PROGRAM PRG1_Conveyer_Operation
VAR_INPUT
	
END_VAR
VAR
	weegTijd 			: INT 			:= 0;
	weegEind 			: INT 			:= 50;
	runningTijd  		: INT 			:= 0;
	detectieLaagTijd  	: INT 			:= 40;
	alarmTijd			: INT			:= 0;
	Modus				: STRING(INT#8) := 'OFF';
	voortangDeling		: INT			:= 100;
	checkpunt			: INT 			:= 0;
END_VAR


// Read startknop
IF NOT GVL.KN_001 AND NOT GVL.alarmActief THEN
	GVL.PRG1_Status := 0;
	GVL.transportActief := FALSE;
END_IF

//als alarm dan naar FAULT
IF NOT GVL.KN_001 AND GVL.alarmActief THEN
	GVL.PRG1_Status := 3;
END_IF

//case functie, voor conveyerstatussen
CASE GVL.PRG1_Status OF
	0:	// OFF, wacht op startknop
		Modus := 'OFF';
		
		IF GVL.KN_001 THEN
			GVL.PRG1_Status := 1;
		END_IF
	1: // idle, wacht op object	
		Modus := 'IDLE';
		
		//reset berekening voor volgende weging
		GVL.berekendeSnelheid := 0;
		
		// als no object detected berekent FC1 de maximale tijd tot alarm
		IF GVL.objectDetected = TRUE THEN
			
			weegTijd := weegTijd + 2;
			GVL.ladingGewicht := GVL.weegcelWaarde;								
			GVL.berekendeSnelheid := FC1_Bereken_Snelheid(GVL.ladingGewicht);//GVL.MinGewicht, GVL.MaxGewicht,GVL.MinSpeed,GVL.MaxSpeed
			IF weegTijd >= weegEind THEN
				GVL.PRG1_Status := 2;
				//reset weegtijd
				weegTijd := 0;
			END_IF
			
		END_IF
		
	2: //running
		Modus := 'RUNNING';
		
		GVL.transportActief := TRUE;
		GVL.geschrevenSnelheid := GVL.berekendeSnelheid;
			
		// Runtijd tellen
		runningTijd := runningTijd + 10;
		
		IF runningTijd > 4 THEN // reset sensor
			GVL.LS_001 := FALSE;
		END_IF
		
		// Tijd conversie naar transportbaan voortgang.
		GVL.transportBaanVoortgang := GVL.geschrevenSnelheid * (runningTijd/voortangDeling);
		
		// Vergelijk voortgang met einde transportbaan, vervolgens reset waarden en status naar IDLE
		IF GVL.transportBaanVoortgang >= GVL.transportBaanEinde THEN
			GVL.transportActief := FALSE;
			GVL.transportBaanVoortgang := 0;
			GVL.geschrevenSnelheid := 0; 
			runningTijd := 0;
			GVL.PRG1_Status := 1;
		END_IF
		
	3: // Fault
		Modus := 'FAULT';
		IF GVL.KN_002 THEN
			GVL.alarmActief := FALSE;
			GVL.PRG1_Status := 1;
		END_IF
END_CASE

END_PROGRAM

(* stored: Version 1.1.0.1, ProductVersion 3.1.4024.12
   POU PRG1_Conveyer_Operation: Id {fa1e73bd-a5a7-4194-991b-8213e2bc5537}, SpecialFunc None *)
